{attribute 'qualified_only'}
{attribute 'strict'}
TYPE E_kierunek :
(
	lewo:=1,
	dol,
	prawo,
	gora
);
END_TYPE

(* stored: Version 1.1.0.1, ProductVersion 3.1.4024.4
   DUT E_kierunek: Id {a27e1feb-095a-4e74-999e-39e516c03d4f} *)
